// TwinCAT 3 PLC project VFFS
// ProgramVersion: 3.1.4026.27
// CompilerDefines: VISU_USEPROPERTYINFO
// libraries:
//   [ApplicationBase], * (Beckhoff Automation LLC)
//   Tc2_EtherCAT, * (Beckhoff Automation GmbH)
//   Tc2_Standard, * (Beckhoff Automation GmbH)
//   Tc2_System, * (Beckhoff Automation GmbH)
//   Tc3_Mc3Ptp, * (Beckhoff Automation GmbH)
//   Tc3_PackML_V3, * (Beckhoff Automation GmbH)
// project tree:
//   / MAIN.TcPOU, PlcTask.TcTTO
//   PullWheel %28EM%29/Interface/ I_PullWheels.TcIO (not stored)
//   PullWheel %28EM%29/ PullWheels.TcPOU (not stored)
//   Sealer %28EM%29/Interface/ I_Sealer.TcIO (not stored)
//   Sealer %28EM%29/ Sealer.TcPOU (not stored), Sealer_TcEvents.TcPOU (not stored)
//   Unwind %28EM%29/Interface/ I_Unwind.TcIO (not stored)
//   Unwind %28EM%29/ Unwind.TcPOU (not stored)
//   VFFS %28MM%29/DUT/ ST_AxisRecipe.TcDUT (not stored), ST_PullWheelsRecipe.TcDUT (not stored), ST_Recipe.TcDUT (not stored), ST_SealerRecipe.TcDUT (not stored), ST_UnwindRecipe.TcDUT (not stored), ST_VFFS_HMI.TcDUT (not stored)
//   VFFS %28MM%29/Interface/ I_VFFS.TcIO (not stored)
//   VFFS %28MM%29/ VFFS.TcPOU (not stored), VFFS_HMI.TcPOU (not stored)
//   Visu/ GlobalTextList.TcGTLO, Visualization Manager.TcVMO (not stored), V_Main.TcVIS
//   Visu/User Controls/ V_PackMLModule.TcVIS
//   _Components/Custom Hmi/ Custom_HMI.TcPOU
//   _Components/Custom Hmi/DUT/ ST_Custom_HMI.TcDUT
//   _Components/Seal Bar/ I_SealBar.TcIO, SealBar.TcPOU
// (motion and I/O tree: see PLC project unittests)
// real-time tasks:
//   TASK UnitTestsBase: cycle T#10ms, priority 20, ADS port 350
//   TASK VFFS: cycle T#10ms, priority 21, ADS port 351
//   TASK PlcTask: cycle T#10ms, priority 22, ADS port 352
//   TASK Job Task: cycle default, priority 32
//   TASK MC-Task (MET): cycle T#2ms, priority 3, ADS port 521
//   TASK MC-Task (MPT): cycle T#10ms, priority 9, ADS port 531
// variable links:

CONFIGURATION VFFS
    RESOURCE PLC ON TwinCAT3
        TASK PlcTask(INTERVAL := T#10ms, PRIORITY := 21);
        PROGRAM MAIN WITH PlcTask : MAIN;
    END_RESOURCE
END_CONFIGURATION

// ---- _Components/Custom Hmi/DUT/ST_Custom_HMI.TcDUT
TYPE ST_Custom_HMI EXTENDS ST_HmiFunction :
	STRUCT
	END_STRUCT
END_TYPE

// ---- _Components/Seal Bar/I_SealBar.TcIO
INTERFACE I_SealBar EXTENDS I_Component

{attribute 'monitoring' := 'call'}
PROPERTY ActualTemperature : LREAL
GET
END_GET
END_PROPERTY

{attribute 'monitoring' := 'call'}
PROPERTY Heat : BOOL
GET
END_GET
SET
END_SET
END_PROPERTY

{attribute 'monitoring' := 'call'}
PROPERTY InTempRange : BOOL
GET
END_GET
END_PROPERTY

{attribute 'monitoring' := 'call'}
PROPERTY SetTemperature : LREAL
GET
END_GET
SET
END_SET
END_PROPERTY

END_INTERFACE

// ---- MAIN.TcPOU
PROGRAM MAIN
VAR
	VFFS		   : VFFS('Vertical from fill Seal');
	MachineHmiTree : GetSystemTreeJsonHmiVisitor<10000>('MAIN');
END_VAR

IF NOT VFFS.Initialized THEN
	VFFS.Initialize();
	MachineHmiTree.GetTree(VFFS);
	RETURN;
END_IF

VFFS.CyclicLogic();

END_PROGRAM

// ---- _Components/Custom Hmi/Custom_HMI.TcPOU
FUNCTION_BLOCK Custom_HMI EXTENDS HmiFunction
VAR
	{ attribute 'TcHmiSymbol.AddSymbol' }
	{ attribute 'TcHmiSymbol.AddSymbol.UserGroups' := '__SystemAdministrators,Admin' }
	Custom_HMI : ST_Custom_HMI;
END_VAR

PROPERTY ControlObject : I_Base
SET
END_SET
END_PROPERTY

METHOD CyclicLogic
Custom_HMI.Name		  := Name;
Custom_HMI.HmiEnabled := Enabled;
END_METHOD

(*FB_Init is always available implicitly and it is used primarily for initialization.
The return value is not evaluated. For a specific influence, you can also declare the
methods explicitly and provide additional code there with the standard initialization
code. You can evaluate the return value.*)
METHOD FB_Init : BOOL
VAR_INPUT
	(* TRUE: the retain variables are initialized (reset warm / reset cold)*)
	bInitRetains : BOOL;

	(* TRUE: the instance will be copied to the copy code afterward (online change)   *)
	bInCopyCode : BOOL;
	Name		: T_MaxString;
END_VAR
ControlType := 'Custom';
LinkObject	:= 'Custom_HMI';
END_METHOD

END_FUNCTION_BLOCK

// ---- _Components/Seal Bar/SealBar.TcPOU
FUNCTION_BLOCK SealBar EXTENDS CyclicComponent IMPLEMENTS I_SealBar
VAR
	_SetTemperature	   : LREAL;
	_ActualTemperature : LREAL;
	_Heat AT %Q*	   : BOOL;
	TempUpdate		   : TON;
	_InTempRange	   : BOOL;
END_VAR

{attribute 'monitoring' := 'call'}
PROPERTY ActualTemperature : LREAL
GET
ActualTemperature := _ActualTemperature;
END_GET
END_PROPERTY

METHOD CyclicLogic
(*Temperature for simulation of temperature changes
This will add 0.3 every 100ms to actual until it gets to Setpoint
It will subtract 0.1 degrees every 100ms unitl it is down to setpoint or 20
Do not set below 20 or it will not get passed resetting*)
TempUpdate(IN := NOT TempUpdate.Q, PT := T#100MS);
IF TempUpdate.Q THEN
	IF _Heat AND _ActualTemperature < _SetTemperature THEN
		_ActualTemperature := _ActualTemperature + 0.3;
	ELSIF _ActualTemperature > 20 THEN
		_ActualTemperature := _ActualTemperature - 0.1;
	END_IF
END_IF

IF ABS(_SetTemperature - _ActualTemperature) < 1 THEN
	_InTempRange := TRUE;
ELSE
	_InTempRange := FALSE;
END_IF
END_METHOD

{attribute 'monitoring' := 'call'}
PROPERTY Heat : BOOL
GET
Heat := _Heat;
END_GET
SET
_Heat := Heat;
END_SET
END_PROPERTY

{attribute 'monitoring' := 'call'}
PROPERTY InTempRange : BOOL
GET
InTempRange := _InTempRange;
END_GET
END_PROPERTY

{attribute 'monitoring' := 'call'}
PROPERTY SetTemperature : LREAL
GET
SetTemperature := _SetTemperature;
END_GET
SET
_SetTemperature := SetTemperature;
END_SET
END_PROPERTY

END_FUNCTION_BLOCK

// ---- Visu/GlobalTextList.TcGTLO
TEXTLIST GlobalTextList
  334 = '%s'
  874 = 'Abort'
  724 = 'Clear'
  690 = 'Complete'
  358 = 'Current Mode: %s'
  446 = 'Current State: %s'
  256 = 'E-Stop Active'
  793 = 'E-Stop OK'
  213 = 'Hold'
  75 = 'Maintenance'
  105 = 'Manual'
  624 = 'Part Time: %2.2f s'
  235 = 'Parts Produced: %d'
  648 = 'Production'
  530 = 'Pulling Time: %2.2f s'
  96 = 'Reset'
  935 = 'Seal act Temp: %3.2f'
  939 = 'Seal set Temp: %3.2f'
  838 = 'Sealing Time: %2.2f s'
  352 = 'Start'
  365 = 'Stop'
  732 = 'Suspend'
  152 = 'Unhold'
  225 = 'Unsuspend'
END_TEXTLIST

// ---- Visu/User Controls/V_PackMLModule.TcVIS
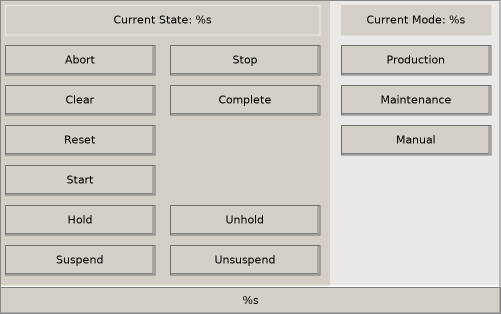
VISUALIZATION V_PackMLModule  // 501x314
VAR_IN_OUT
	PackML_HMI : ST_PackMLStatemachine_HMI;
END_VAR
    Rectangle (0,0 330x285)
    Textfield (5,5 315x30), "Current State: %s", text variable: PackML_HMI.CurrentState
    Button (5,45 150x30), "Abort"
        OnMouseClick: execute { PackML_HMI.StateCommand := E_PMLCommand.Abort; }
    Button (5,85 150x30), "Clear"
        OnMouseClick: execute { PackML_HMI.StateCommand := E_PMLCommand.Clear; }
    Button (5,125 150x30), "Reset"
        OnMouseClick: execute { PackML_HMI.StateCommand := E_PMLCommand.Reset; }
    Button (5,165 150x30), "Start"
        OnMouseClick: execute { PackML_HMI.StateCommand := E_PMLCommand.Start; }
    Button (170,85 150x30), "Complete"
        OnMouseClick: execute { PackML_HMI.StateCommand := E_PMLCommand.Complete; }
    Button (170,45 150x30), "Stop"
        OnMouseClick: execute { PackML_HMI.StateCommand := E_PMLCommand.Stop; }
    Button (5,205 150x30), "Hold"
        OnMouseClick: execute { PackML_HMI.StateCommand := E_PMLCommand.Hold; }
    Button (170,205 150x30), "Unhold"
        OnMouseClick: execute { PackML_HMI.StateCommand := E_PMLCommand.Unhold; }
    Button (5,245 150x30), "Suspend"
        OnMouseClick: execute { PackML_HMI.StateCommand := E_PMLCommand.Suspend; }
    Button (170,245 150x30), "Unsuspend"
        OnMouseClick: execute { PackML_HMI.StateCommand := E_PMLCommand.Unsuspend; }
    Rectangle (330,0 171x285)
    Textfield (341,5 150x30), "Current Mode: %s", text variable: PackML_HMI.CurrentMode
    Button (341,45 150x30), "Production"
        OnMouseClick: execute { PackML_HMI.ModeCommand := 1; }
    Button (341,85 150x30), "Maintenance"
        OnMouseClick: execute { PackML_HMI.ModeCommand := 2; }
    Button (341,125 150x30), "Manual"
        OnMouseClick: execute { PackML_HMI.ModeCommand := 3; }
    Textfield (0,287 501x27), "%s", text variable: PackML_HMI.Name
END_VISUALIZATION

// ---- Visu/V_Main.TcVIS
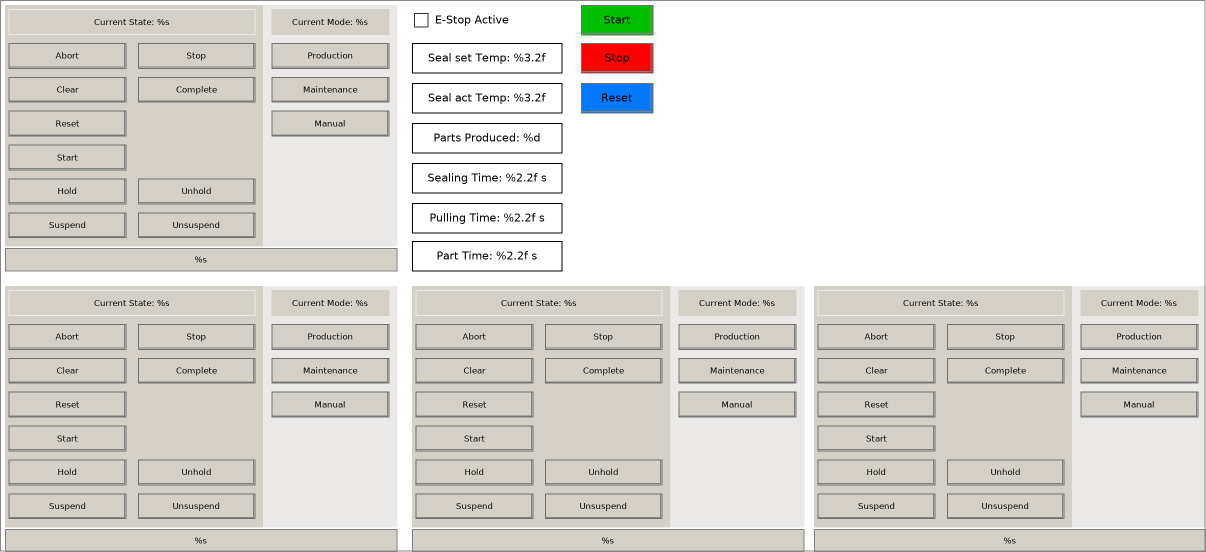
VISUALIZATION V_Main  // 1206x552
    Checkbox (412,5 150x30), "E-Stop Active", variable: MAIN.VFFS.EStop1_Pressed
    Frame (5,5 392x266)
        shows V_PackMLModule(PackML_HMI := MAIN.VFFS.VFFS_HMI.Statemachine_HMI)
    Frame (5,286 392x266)
        shows V_PackMLModule(PackML_HMI := MAIN.VFFS._PullWheels.Statemachine_HMI.Statemachine_HMI)
    Frame (412,286 392x266)
        shows V_PackMLModule(PackML_HMI := MAIN.VFFS._Sealer.Statemachine_HMI.Statemachine_HMI)
    Frame (814,286 392x266)
        shows V_PackMLModule(PackML_HMI := MAIN.VFFS._Unwind.Statemachine_HMI.Statemachine_HMI)
    Rectangle (412,43 150x30), "Seal set Temp: %3.2f", text variable: MAIN.VFFS._Sealer._SealBar._SetTemperature
    Rectangle (412,83 150x30), "Seal act Temp: %3.2f", text variable: MAIN.VFFS._Sealer._SealBar._ActualTemperature
    Rectangle (412,123 150x30), "Parts Produced: %d", text variable: MAIN.VFFS._PartsProduced
    Button (581,5 72x30), "Start", input disabled if: NOT MAIN.VFFS.VFFS_HMI.Statemachine_HMI.StartPermissive
        OnMouseDown: execute { MAIN.VFFS.VFFS_HMI.Statemachine_HMI.StartPressed := TRUE; }
        OnMouseUp: execute { MAIN.VFFS.VFFS_HMI.Statemachine_HMI.StartPressed := FALSE; }
    Button (581,43 72x30), "Stop", input disabled if: NOT MAIN.VFFS.VFFS_HMI.Statemachine_HMI.StopPermissive
        OnMouseDown: execute { MAIN.VFFS.VFFS_HMI.Statemachine_HMI.StopPressed := TRUE; }
        OnMouseUp: execute { MAIN.VFFS.VFFS_HMI.Statemachine_HMI.StopPressed := False; }
    Button (581,83 72x30), "Reset", input disabled if: NOT MAIN.VFFS.VFFS_HMI.Statemachine_HMI.ResetPermissive
        OnMouseDown: execute { MAIN.VFFS.VFFS_HMI.Statemachine_HMI.ResetPressed := TRUE; }
        OnMouseUp: execute { MAIN.VFFS.VFFS_HMI.Statemachine_HMI.ResetPressed := FALSE; }
    Rectangle (412,163 150x30), "Sealing Time: %2.2f s", text variable: MAIN.VFFS._SealingTime
    Rectangle (412,203 150x30), "Pulling Time: %2.2f s", text variable: MAIN.VFFS._PullingTime
    Rectangle (412,241 150x30), "Part Time: %2.2f s", text variable: MAIN.VFFS._PartTime
END_VISUALIZATION
